% RSLogix 500 project I2P-Job16-Adam Boczkiewicz.RSS, saved by version 10.00.00.00 %
PROJECT "ML04A"    % processor: Bul.1763 MicroLogix 1100 Series B %

PROGRAM FILES
  LAD 2   6 rungs

DATA FILES
  O0 OUTPUT  4 elements
  I1 INPUT  6 elements
  S2 STATUS  66 elements
  B3 BINARY  1 elements
  T4 TIMER  1 elements
  C5 COUNTER  1 elements
  R6 CONTROL  1 elements
  N7 INTEGER  1 elements
  F8 FLOAT  1 elements

LADDER 2
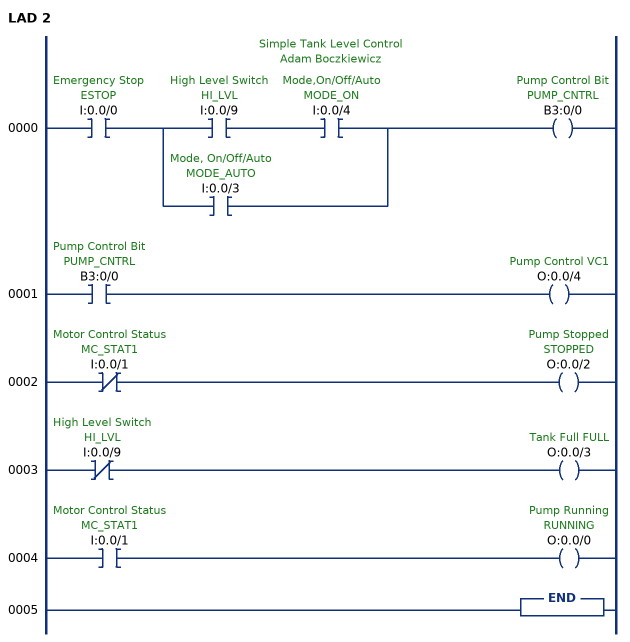
% Rung: 0 %
% Simple Tank Level Control
% Adam Boczkiewicz %
SOR XIC I:0.0/0 BST XIC I:0.0/9 XIC I:0.0/4 NXB XIC I:0.0/3 BND OTE B3:0/0 EOR
%   I:0.0/0  ESTOP  "Emergency Stop" %
%   I:0.0/9  HI_LVL  "High Level Switch" %
%   I:0.0/4  MODE_ON  "Mode,On/Off/Auto" %
%   I:0.0/3  MODE_AUTO  "Mode, On/Off/Auto" %
%   B3:0/0  PUMP_CNTRL  "Pump Control Bit" %
% Rung: 1 %
SOR XIC B3:0/0 OTE O:0.0/4 EOR
%   B3:0/0  PUMP_CNTRL  "Pump Control Bit" %
%   O:0.0/4  VC1  "Pump Control" %
% Rung: 2 %
SOR XIO I:0.0/1 OTE O:0.0/2 EOR
%   I:0.0/1  MC_STAT1  "Motor Control Status" %
%   O:0.0/2  STOPPED  "Pump Stopped" %
% Rung: 3 %
SOR XIO I:0.0/9 OTE O:0.0/3 EOR
%   I:0.0/9  HI_LVL  "High Level Switch" %
%   O:0.0/3  FULL  "Tank Full" %
% Rung: 4 %
SOR XIC I:0.0/1 OTE O:0.0/0 EOR
%   I:0.0/1  MC_STAT1  "Motor Control Status" %
%   O:0.0/0  RUNNING  "Pump Running" %
% Rung: 5 %
SOR END EOR

OTHER DOCUMENTED ADDRESSES
  B3:0/1  JBR  "Jog Bit Reverse"
  B3:0/2  FB  "Foward Bit"
  B3:0/3  RB  "Reverse Bit"
  B3:0/4  DCF  "Last Direction Foward Bit"
  B3:0/5  DCR  "Last Direction Reverse Bit"
  B3:0/6  YB  "Yellow Bit"
  I:0.0/2  DIR_STAT1  "Motor Direction Status"
  I:0.0/5  OFF_AUTO  "Off Or Auto"
  I:0.0/6  STOP  "Stop Motor"
  I:0.0/7  START  "Start Motor"
  I:0.0/8  REV  "Jog Motor"
  JOG  
  MO  
  O:0.0/1  AUTO  "Auto Control"
  O:0.0/5  CR2  "Direction Control Relay"
  T4:0/TT  TT

DATA TABLE (non-zero values as saved)
DATA T4
% .PRE .ACC %
% T4:0 % 8 0
DATA C5
% .PRE .ACC %
% C5:0 % 16 1
